(* IEC 61131-3 sources: Industry-PLC-LLM/data/PLCBEAD_repo/PLCBEAD_PLCEmbed-main/PLC-BEAD/Source/GEB/V3_SUB, 1 file *)

(* ---- V3_SUB.ST ---- *)
TYPE oscat_vector_3:
	STRUCT
		X : REAL;
		Y : REAL;
		Z : REAL;
	END_STRUCT;
END_TYPE

FUNCTION_BLOCK V3_SUB_Block

	VAR_INPUT
		A :	oscat_vector_3;
		B :	oscat_vector_3;
	END_VAR

	VAR_OUTPUT
		V3_SUB :	oscat_vector_3;
	END_VAR

	V3_SUB.X := A.X - B.X;
	V3_SUB.Y := A.Y - B.Y;
	V3_SUB.Z := A.Z - B.Z;

END_FUNCTION_BLOCK

PROGRAM program0
  	VAR
		A :	oscat_vector_3;
		B :	oscat_vector_3;
		V3_SUB :	oscat_vector_3;
		func_block : V3_SUB_Block;
  	END_VAR
	func_block.A := A;
	func_block.B := B;
	func_block();
	V3_SUB := func_block.V3_SUB;
END_PROGRAM
